// TwinCAT 3 PLC project bridge
// ProgramVersion: 3.1.4023.0
// libraries:
//   Tc2_Standard, * (Beckhoff Automation GmbH)
//   Tc2_System, * (Beckhoff Automation GmbH)
//   Tc3_Module, * (Beckhoff Automation GmbH)
// project tree:
//   DUTs/ XinputState.TcDUT, XINPUT_GAMEPAD.TcDUT
//   GVLs/ JSDATA.TcGVL
//   / PlcTask.TcTTO
//   POUs/ MAIN.TcPOU
// real-time tasks:
//   TASK PlcTask: cycle T#10ms, priority 20, ADS port 350

CONFIGURATION bridge
    RESOURCE PLC ON TwinCAT3
        TASK PlcTask(INTERVAL := T#10ms, PRIORITY := 20);
        PROGRAM MAIN WITH PlcTask : MAIN;
    END_RESOURCE
END_CONFIGURATION

// ---- DUTs/XinputState.TcDUT
TYPE XinputState:
STRUCT
	dwPacketNumber :DWORD;
	Gamepad : XINPUT_GAMEPAD;
END_STRUCT
END_TYPE

// ---- DUTs/XINPUT_GAMEPAD.TcDUT
TYPE XINPUT_GAMEPAD :
STRUCT
 wButtons: WORD;
 bLeftTrigger: BYTE;
 bRightTrigger: BYTE;
 sThumbLX: INT;
 sThumbLY: INT;
 sThumbRX: INT;
 sThumbRY: INT;
END_STRUCT
END_TYPE

// ---- GVLs/JSDATA.TcGVL
{attribute 'qualified_only'}
VAR_GLOBAL
GamepadState : XinputState;
END_VAR

// ---- POUs/MAIN.TcPOU
PROGRAM MAIN
VAR
END_VAR

END_PROGRAM
